// TIA Portal project "sequantial_turn_tables_project" (V16)
// Vorlageprojekt für das Buch mit Zielsystem S7-1200

(* hardware
DEVICE "S7-1200-Station_1"  S7-1200 Station
   slot 0: "Baugruppenträger_0"  Rack  V1.0
   slot 1: "PLC_1"  CPU 1211C DC/DC/DC  6ES7 211-1AE40-0XB0  V4.1
*)

// ===== PLC "PLC_1"  CPU 1211C DC/DC/DC =====

VAR_GLOBAL   // PLC tag table "Standard-Variablentabelle"
   "sistem" AT %M0.0 : Bool;
   "Emergency" AT %I1.6 : Bool;
   "Display" AT %QD30 : Real;
   "Curved_Roller_Conveyor" AT %Q1.0 : Bool;
END_VAR

VAR_GLOBAL   // PLC tag table "Tag table from XML_2"
   "sensor_1" AT %I0.0 : Bool;
   "sensor_2" AT %I0.1 : Bool;
   "turntable_0_degree" AT %I0.2 : Bool;
   "turntable_90_degree" AT %I0.3 : Bool;
   "front_limit_sensor" AT %I0.4 : Bool;
   "Start Button 1" AT %I0.5 : Bool;
   "Stop Button 1" AT %I0.6 : Bool;
   "sensor_4" AT %I0.7 : Bool;
   "Diffuse Sensor 3" AT %I1.0 : Bool;
   "Diffuse Sensor 5" AT %I1.1 : Bool;
   "Turntable 2 (Limit 0)" AT %I1.2 : Bool;
   "Turntable 2 (Limit 90)" AT %I1.3 : Bool;
   "Turntable 2 (Front Limit)" AT %I1.4 : Bool;
   "Diffuse Sensor 6" AT %I1.5 : Bool;
   "Roller Conveyor (4m) 1" AT %Q0.0 : Bool;
   "Roller Conveyor (4m) 2" AT %Q0.1 : Bool;
   "Turntable 1 Turn" AT %Q0.2 : Bool;
   "Turntable 1 Roll (+)" AT %Q0.3 : Bool;
   "Roller Conveyor (4m) 3" AT %Q0.4 : Bool;
   "Roller Conveyor (4m) 4" AT %Q0.5 : Bool;
   "Turntable 2 Turn" AT %Q0.6 : Bool;
   "Turntable 2 Roll (+)" AT %Q0.7 : Bool;
END_VAR

DATA_BLOCK "turn_table_DB"   // DB1
{ S7_Optimized_Access := 'TRUE' }
VERSION : 0.1
// stored: InstanceOfName turn_table
"turn_table"
BEGIN
END_DATA_BLOCK

DATA_BLOCK "turn_table_DB_1"   // DB2
{ S7_Optimized_Access := 'TRUE' }
VERSION : 0.1
// stored: InstanceOfName turn_table
"turn_table"
BEGIN
END_DATA_BLOCK

FUNCTION_BLOCK "turn_table"   // FB1, LAD
{ S7_Optimized_Access := 'TRUE' }
VERSION : 0.1
   VAR_INPUT
      sistem : Bool;
      sensor_1 : Bool;
      sensor_2 : Bool;
      turn_table_90_deg : Bool;
      turn_table_0_deg : Bool;
      front_limit_sensor : Bool;
      sensor_4 : Bool;
   END_VAR
   VAR_OUTPUT
      turn_table_turn : Bool;
      roller_conveyor_1 : Bool;
      turn_table_roller : Bool;
      roller_conveyor_2 : Bool;
   END_VAR
BEGIN

REGION Network 1
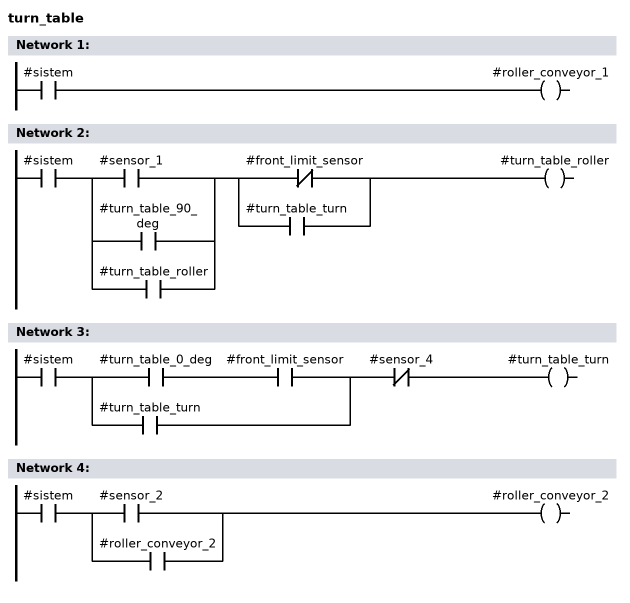
   RUNG wire#powerrail
      Contact( #sistem )
      Coil( #roller_conveyor_1 )
   END_RUNG
   // the same network as SCL:
   #roller_conveyor_1 := #sistem;
END_REGION

REGION Network 2
   RUNG wire#powerrail
      Contact( #sistem )
      wire#w1
      Contact( #sensor_1 )
      wire#w2
      I_Contact( #front_limit_sensor )
      wire#w3
      Coil( #turn_table_roller )
   END_RUNG
   RUNG wire#w1
      Contact( #turn_table_90_deg )
   END_RUNG wire#w2
   RUNG wire#w1
      Contact( #turn_table_roller )
   END_RUNG wire#w2
   RUNG wire#w2
      Contact( #turn_table_turn )
   END_RUNG wire#w3
   // the same network as SCL:
   #turn_table_roller := #sistem AND (#sensor_1 OR #turn_table_90_deg OR #turn_table_roller) AND (NOT #front_limit_sensor OR #turn_table_turn);
END_REGION

REGION Network 3
   RUNG wire#powerrail
      Contact( #sistem )
      wire#w1
      Contact( #turn_table_0_deg )
      Contact( #front_limit_sensor )
      wire#w2
      I_Contact( #sensor_4 )
      Coil( #turn_table_turn )
   END_RUNG
   RUNG wire#w1
      Contact( #turn_table_turn )
   END_RUNG wire#w2
   // the same network as SCL:
   #turn_table_turn := #sistem AND ((#turn_table_0_deg AND #front_limit_sensor) OR #turn_table_turn) AND NOT #sensor_4;
END_REGION

REGION Network 4
   RUNG wire#powerrail
      Contact( #sistem )
      wire#w1
      Contact( #sensor_2 )
      wire#w2
      Coil( #roller_conveyor_2 )
   END_RUNG
   RUNG wire#w1
      Contact( #roller_conveyor_2 )
   END_RUNG wire#w2
   // the same network as SCL:
   #roller_conveyor_2 := #sistem AND (#sensor_2 OR #roller_conveyor_2);
END_REGION
END_FUNCTION_BLOCK

FUNCTION "MHJ-PLC-Lab-Function-S71200" : Void   // FC9000, SCL
{ S7_Optimized_Access := 'TRUE' }
VERSION : 0.1
   VAR_TEMP
      rdTimeReturn : Int;
      outputTime : DTL;
      SyncVal : Byte;
      forVal : Int;
      forVal_2 : Int;
      Value : Byte;
   END_VAR
   VAR CONSTANT
      CompVal : Byte := 16#34;
      Value_01 : Byte := 16#11;
      Value_01_DW : DWord := 16#A165_D992;
      Value_02_DW : DWord := 16#58BE_4401;
   END_VAR
BEGIN

   #Value:=PEEK(area := 16#82,
        dbNumber := 0,
        byteOffset := 511);
   #Value := #Value + 1;

   POKE(area := 16#82,
        dbNumber := 0,
        byteOffset := 511,
        value := #Value);

   POKE(area:=16#81,
        dbNumber:=0,
        byteOffset:=1016,
        value:=#Value_01_DW);
   POKE(area := 16#81,
        dbNumber := 0,
        byteOffset := 1020,
        value := #Value_02_DW);

   POKE(area := 16#81,
        dbNumber := 0,
        byteOffset := 511,
        value := B#16#00);

   FOR #forVal := 0 TO 120 DO
       FOR #forVal_2:=0 TO 10 DO
           #rdTimeReturn:=RD_SYS_T(#outputTime);
           #rdTimeReturn := WR_SYS_T(#outputTime);
           #rdTimeReturn := RD_SYS_T(#outputTime);
           #rdTimeReturn := WR_SYS_T(#outputTime);
       END_FOR;
       #SyncVal:= PEEK(area := 16#81,
                      dbNumber := 0,
                      byteOffset := 511);
       IF #SyncVal = #CompVal THEN
          GOTO M_1;
       END_IF;
   END_FOR;
   RETURN;

   M_1:
   POKE(area := 16#81,
        dbNumber := 0,
        byteOffset := 511,
        value := B#16#0);
END_FUNCTION

ORGANIZATION_BLOCK "Main"   // OB1, LAD, ProgramCycle
TITLE = "Main Program Sweep (Cycle)"
{ S7_Optimized_Access := 'TRUE' }
VERSION : 0.1
   VAR_INPUT
      Initial_Call : Bool;   // Initial call of this OB
      Remanence : Bool;   // =True, if remanent data are available
   END_VAR
BEGIN

REGION Network 1: Konnektierungsbaustein für PLC-Lab
   // Im Netzwerk 1 wird der Konnektierungsbaustein für PLC-Lab aufgerufen.
   // Dieser Aufruf darf nicht entfernt werden!
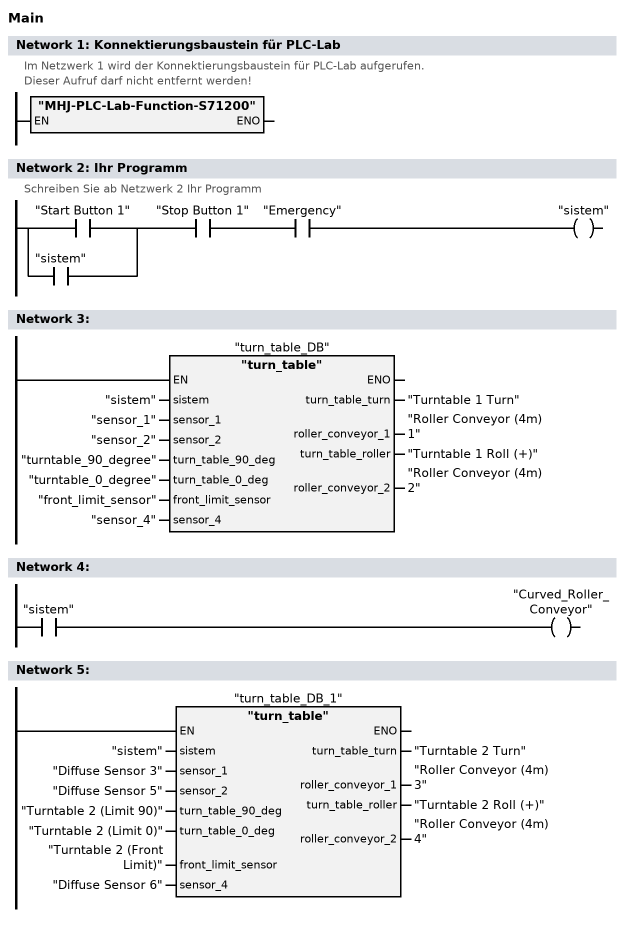
   RUNG wire#powerrail
      "MHJ-PLC-Lab-Function-S71200"()
   END_RUNG
   // the same network as SCL:
   "MHJ-PLC-Lab-Function-S71200"();
END_REGION

REGION Network 2: Ihr Programm
   // Schreiben Sie ab Netzwerk 2 Ihr Programm
   RUNG wire#powerrail
      Contact( "Start Button 1" )
      wire#w1
      Contact( "Stop Button 1" )
      Contact( "Emergency" )
      Coil( "sistem" )
   END_RUNG
   RUNG wire#powerrail
      Contact( "sistem" )
   END_RUNG wire#w1
   // the same network as SCL:
   "sistem" := ("Start Button 1" OR "sistem") AND "Stop Button 1" AND "Emergency";
END_REGION

REGION Network 3
   RUNG wire#powerrail
      "turn_table_DB"(sistem := "sistem", sensor_1 := "sensor_1", sensor_2 := "sensor_2", turn_table_90_deg := "turntable_90_degree", turn_table_0_deg := "turntable_0_degree", front_limit_sensor := "front_limit_sensor", sensor_4 := "sensor_4", turn_table_turn => "Turntable 1 Turn", roller_conveyor_1 => "Roller Conveyor (4m) 1", turn_table_roller => "Turntable 1 Roll (+)", roller_conveyor_2 => "Roller Conveyor (4m) 2")
   END_RUNG
   // the same network as SCL:
   "turn_table_DB"(sistem := "sistem",   // "turn_table"
                   sensor_1 := "sensor_1",
                   sensor_2 := "sensor_2",
                   turn_table_90_deg := "turntable_90_degree",
                   turn_table_0_deg := "turntable_0_degree",
                   front_limit_sensor := "front_limit_sensor",
                   sensor_4 := "sensor_4",
                   turn_table_turn => "Turntable 1 Turn",
                   roller_conveyor_1 => "Roller Conveyor (4m) 1",
                   turn_table_roller => "Turntable 1 Roll (+)",
                   roller_conveyor_2 => "Roller Conveyor (4m) 2");
END_REGION

REGION Network 4
   RUNG wire#powerrail
      Contact( "sistem" )
      Coil( "Curved_Roller_Conveyor" )
   END_RUNG
   // the same network as SCL:
   "Curved_Roller_Conveyor" := "sistem";
END_REGION

REGION Network 5
   RUNG wire#powerrail
      "turn_table_DB_1"(sistem := "sistem", sensor_1 := "Diffuse Sensor 3", sensor_2 := "Diffuse Sensor 5", turn_table_90_deg := "Turntable 2 (Limit 90)", turn_table_0_deg := "Turntable 2 (Limit 0)", front_limit_sensor := "Turntable 2 (Front Limit)", sensor_4 := "Diffuse Sensor 6", turn_table_turn => "Turntable 2 Turn", roller_conveyor_1 => "Roller Conveyor (4m) 3", turn_table_roller => "Turntable 2 Roll (+)", roller_conveyor_2 => "Roller Conveyor (4m) 4")
   END_RUNG
   // the same network as SCL:
   "turn_table_DB_1"(sistem := "sistem",   // "turn_table"
                     sensor_1 := "Diffuse Sensor 3",
                     sensor_2 := "Diffuse Sensor 5",
                     turn_table_90_deg := "Turntable 2 (Limit 90)",
                     turn_table_0_deg := "Turntable 2 (Limit 0)",
                     front_limit_sensor := "Turntable 2 (Front Limit)",
                     sensor_4 := "Diffuse Sensor 6",
                     turn_table_turn => "Turntable 2 Turn",
                     roller_conveyor_1 => "Roller Conveyor (4m) 3",
                     turn_table_roller => "Turntable 2 Roll (+)",
                     roller_conveyor_2 => "Roller Conveyor (4m) 4");
END_REGION
END_ORGANIZATION_BLOCK